(* IEC 61131-3 sources: std_i2980_v2.06_cp053/Source/IMM/ieccontrol/HostCommunication (part 2) *)

(* ---- FTimeToSec.pu ---- *)
(*
@h    ! WARNING !
@h    The Kemro K2 system (including software) only meets category B according to EN 954-1,
@h    thus it is not intended for usage in safety-relevant control applications in the field
@h    of personal safety (e.g. emergency stop).
@h    To implement potentially necessary safety-relevant control tasks, always use additional
@h    external safety devices that are intended for the particular purpose, and meet the necessary
@h    functional safety.
@h    For further information see EN 954-1 (EN ISO 13849-1) and/or the K2-x00 user manual, chapter
@h    "CE conformity, directives and standards".

returns a REAL value (unit s, precision 3 digits after point) for a TIME value

*)

FUNCTION FTimeToSec : REAL #DUMMY_EDIT_BLOCK

VAR_INPUT
 time : TIME;
END_VAR
#BEGIN_EDIT_BLOCK
(**************************************** WARNING ********************************************
 *** The KEBA Kemro K2 System including software is not intended for safety control tasks! ***
 ***                       For further information see Comment tab!                        ***
 *********************************************************************************************)

FTimeToSec := LINT_TO_REAL((TIME_TO_LINT(time)/1000))/1000.0;

;#END_EDIT_BLOCK END_FUNCTION

#END_OF_IEC_PART

@Puma @IecEditor 6 60 @Pou 25
@@@BEG_Comment@@@
@h    ! WARNING !
@h    The Kemro K2 system (including software) only meets category B according to EN 954-1,
@h    thus it is not intended for usage in safety-relevant control applications in the field
@h    of personal safety (e.g. emergency stop).
@h    To implement potentially necessary safety-relevant control tasks, always use additional
@h    external safety devices that are intended for the particular purpose, and meet the necessary
@h    functional safety.
@h    For further information see EN 954-1 (EN ISO 13849-1) and/or the K2-x00 user manual, chapter
@h    "CE conformity, directives and standards".

returns a REAL value (unit s, precision 3 digits after point) for a TIME value

@@@END_Comment@@@

@BEG_Contents

@BEG_Func
@RT(17)FuncTreeContainer
0
@END_Func

@BEG_Const
@RT(18)ConstTreeContainer
0
@END_Const

@BEG_Export

@BEG_Kind
@FUNCTION @RT(10)FTimeToSec @STRUCTURED_TEXT
@RT(4)REAL @RT(0) @RT(0)
@END_Kind

@BEG_Dcl
@RT(16)DclTreeContainer
1
@Var @RT(4)time @RT(0) @T @F @DT @RT(4)TIME @RT(0) @T @T @BASIC 0 @F
@F @F
@T
@BEG_Attrib
3 @RT(0) @RT(0) @RT(0)
@END_Attrib
1 1 @F @F @F @F

@END_Dcl

@END_Export

@BEG_Body
@TL(7)
(**************************************** WARNING ********************************************
 *** The KEBA Kemro K2 System including software is not intended for safety control tasks! ***
 ***                       For further information see Comment tab!                        ***
 *********************************************************************************************)

FTimeToSec := LINT_TO_REAL((TIME_TO_LINT(time)/1000))/1000.0;

@END_Body

@END_Contents

(* ---- ABEM63.pu ---- *)
(*
@h    ! WARNING !
@h    The Kemro K2 system (including software) only meets category B according to EN 954-1,
@h    thus it is not intended for usage in safety-relevant control applications in the field
@h    of personal safety (e.g. emergency stop).
@h    To implement potentially necessary safety-relevant control tasks, always use additional
@h    external safety devices that are intended for the particular purpose, and meet the necessary
@h    functional safety.
@h    For further information see EN 954-1 (EN ISO 13849-1) and/or the K2-x00 user manual, chapter
@h    "CE conformity, directives and standards".

Euromap63 specific application parameters
*)

IMPORT_OVER_LISTFILE
 STOP_PROCESS_ALGORITHM
, GET_SYNC_REFTO
, ASCII_TO_STRING
, cMaxInjectionUnits
, cMaxZones
, tsEM63
, tnOperationMode
, ABHeatingState

END_IMPORT

ALGORITHM_BLOCK ABEM63 #DUMMY_EDIT_BLOCK

SYSTEM_VAR
 sv_EM63 : tsEM63;
 sv_iPendingAlarms : DINT (* number of alarms pending with class 1,2,3 *);
 sv_OperationMode : tnOperationMode;
 sv_bBadPart : BOOL;
 sv_iShotCounterRetain : UDINT (* shot counter retain (used for lubrication) *);
 sv_bInitDone : BOOL (* IEC initialisation is finished (after movement registration) *);
END_VAR

SYSTEM_OBJECT
 TaskVis : TASK;
 PU_Task_7 : TASK;
END_OBJECT

VAR
 mbLastCycleBad : BOOL;
 mpiTrigger : REFTO UDINT;
END_VAR

POSTUPDATE_ALGORITHM pActivate ON TaskVis WITH sv_bInitDone,sv_EM63.bActivate

#BEGIN_EDIT_BLOCK
(**************************************** WARNING ********************************************
 *** The KEBA Kemro K2 System including software is not intended for safety control tasks! ***
 ***                       For further information see Comment tab!                        ***
 *********************************************************************************************)

IF (sv_EM63.bActivate AND sv_bInitDone) THEN
    mpiTrigger := @sv_iShotCounterRetain;
    START_PROCESS_ALGORITHM(paRun);
ELSE
    mpiTrigger := EMPTY;
    STOP_PROCESS_ALGORITHM(paRun);
END_IF;

;#END_EDIT_BLOCK END_ALGORITHM

ALGORITHM aMachineStatus

VAR
 bAlarms : BOOL;
 sMachineMode : STRING(2);
 bActStsChanged : BOOL;
 oldOpMode : tnOperationMode;
 oldAlarms : BOOL;
 oldCycleBad : BOOL;
 bInit : BOOL;
END_VAR
#BEGIN_EDIT_BLOCK
(**************************************** WARNING ********************************************
 *** The KEBA Kemro K2 System including software is not intended for safety control tasks! ***
 ***                       For further information see Comment tab!                        ***
 *********************************************************************************************)

// ActStsMachine
bAlarms := sv_iPendingAlarms > 0;

bActStsChanged := (oldOpMode <> sv_OperationMode) OR (oldAlarms <> bAlarms) OR (oldCycleBad <> mbLastCycleBad);

oldOpMode := sv_OperationMode;
oldAlarms := bAlarms;
oldCycleBad := mbLastCycleBad;

IF (bActStsChanged OR (NOT bInit)) THEN
    bInit := TRUE;

    CASE (sv_OperationMode) OF
        nFullAutomatic: sMachineMode := "A";
        nHalfAutomatic: sMachineMode := "S";
        nManual: sMachineMode := "M";
        nSetup: sMachineMode := "U";
    ELSE
        sMachineMode := "0";
    END_CASE;

    sv_EM63.ActStsMachine := CONCAT("0", sMachineMode, "0", DINT_TO_STRING(BOOL_TO_DINT(mbLastCycleBad)),  DINT_TO_STRING(BOOL_TO_DINT(bAlarms)));
END_IF;

;#END_EDIT_BLOCK END_ALGORITHM

PROCESS_ALGORITHM paRun ON TaskVis

VAR
 iRedCnt : INT;
 abHeatingState : ABHeatingState;
END_VAR
#BEGIN_EDIT_BLOCK
(**************************************** WARNING ********************************************
 *** The KEBA Kemro K2 System including software is not intended for safety control tasks! ***
 ***                       For further information see Comment tab!                        ***
 *********************************************************************************************)

IF (iRedCnt = 0) THEN
   iRedCnt := 5;

   aMachineStatus();
   abHeatingState.aHeating(bEM63 := TRUE);
END_IF;

iRedCnt := iRedCnt - 1;

;#END_EDIT_BLOCK END_ALGORITHM

POSTUPDATE_ALGORITHM pShotCounter ON PU_Task_7(1) WITH mpiTrigger^

#BEGIN_EDIT_BLOCK
(**************************************** WARNING ********************************************
 *** The KEBA Kemro K2 System including software is not intended for safety control tasks! ***
 ***                       For further information see Comment tab!                        ***
 *********************************************************************************************)

mbLastCycleBad := sv_bBadPart;

;#END_EDIT_BLOCK END_ALGORITHM

END_ALGORITHM_BLOCK

#END_OF_IEC_PART

@Puma @IecEditor 6 159 @Pou 25
@@@BEG_Comment@@@
@h    ! WARNING !
@h    The Kemro K2 system (including software) only meets category B according to EN 954-1,
@h    thus it is not intended for usage in safety-relevant control applications in the field
@h    of personal safety (e.g. emergency stop).
@h    To implement potentially necessary safety-relevant control tasks, always use additional
@h    external safety devices that are intended for the particular purpose, and meet the necessary
@h    functional safety.
@h    For further information see EN 954-1 (EN ISO 13849-1) and/or the K2-x00 user manual, chapter
@h    "CE conformity, directives and standards".

Euromap63 specific application parameters
@@@END_Comment@@@

@BEG_Contents

@BEG_Func
@RT(17)FuncTreeContainer
3
@Var @RT(22)STOP_PROCESS_ALGORITHM @RT(0) @T @T @DERIVED 0 @F @RT(23)KEBA_STANDARD_PROCEDURE @F
@T
@BEG_Attrib
0 @RT(0) @RT(0)
@END_Attrib
1 1 @F @F @F @F

@Var @RT(14)GET_SYNC_REFTO @RT(0) @T @T @DERIVED 0 @F @RT(22)KEBA_STANDARD_FUNCTION @F
@T
@BEG_Attrib
0 @RT(0) @RT(0)
@END_Attrib
1 1 @F @F @F @F

@Var @RT(15)ASCII_TO_STRING @RT(0) @T @T @DERIVED 0 @F @RT(22)KEBA_STANDARD_FUNCTION @F
@T
@BEG_Attrib
0 @RT(0) @RT(0)
@END_Attrib
1 1 @F @F @F @F

@END_Func

@BEG_Const
@RT(18)ConstTreeContainer
2
@Var @RT(18)cMaxInjectionUnits @RT(0) @T @F @DT @RT(4)DINT @RT(0) @T @T @BASIC 0 @F
@F @F
@T
@BEG_Attrib
0 @RT(1)2 @RT(0)
@END_Attrib
1 1 @F @F @F @F

@Var @RT(9)cMaxZones @RT(0) @T @F @DT @RT(4)DINT @RT(0) @T @T @BASIC 0 @F
@F @F
@T
@BEG_Attrib
0 @RT(2)72 @RT(27)max number of heating zones
@END_Attrib
1 1 @F @F @F @F

@END_Const

@BEG_Export

@BEG_Kind
@ALGORITHM_BLOCK @RT(6)ABEM63 @STRUCTURED_TEXT
@RT(0) @RT(0) @RT(0)
@END_Kind

@BEG_Dcl
@RT(16)DclTreeContainer
10
@Var @RT(7)sv_EM63 @RT(0) @T @T @DERIVED 0 @F @RT(6)tsEM63 @F
@T
@BEG_Attrib
3 @RT(0) @RT(0) @RT(0)
@END_Attrib
1 8 @F @F @F @F

@Var @RT(17)sv_iPendingAlarms @RT(0) @T @F @DT @RT(4)DINT @RT(0) @T @T @BASIC 0 @F
@F @F
@T
@BEG_Attrib
3 @RT(0) @RT(41)number of alarms pending with class 1,2,3 @RT(0)
@END_Attrib
1 8 @F @F @F @F

@Var @RT(16)sv_OperationMode @RT(0) @T @T @DERIVED 0 @T @T @DT @RT(15)tnOperationMode @RT(0) @T @T @UNKNOWN 0 @F
@F @F
@T
@BEG_Attrib
3 @RT(0) @RT(0) @RT(0)
@END_Attrib
1 8 @F @F @F @F

@Var @RT(11)sv_bBadPart @RT(0) @T @F @DT @RT(4)BOOL @RT(0) @T @T @BASIC 0 @F
@F @F
@T
@BEG_Attrib
3 @RT(0) @RT(0) @RT(0)
@END_Attrib
1 8 @F @F @F @F

@Var @RT(21)sv_iShotCounterRetain @RT(0) @T @F @DT @RT(5)UDINT @RT(0) @T @T @BASIC 0 @F
@F @F
@T
@BEG_Attrib
3 @RT(0) @RT(42)shot counter retain (used for lubrication) @RT(0)
@END_Attrib
1 8 @F @F @F @F

@Var @RT(12)sv_bInitDone @RT(0) @T @F @DT @RT(4)BOOL @RT(0) @T @T @BASIC 0 @F
@F @F
@T
@BEG_Attrib
3 @RT(0) @RT(60)IEC initialisation is finished (after movement registration) @RT(0)
@END_Attrib
1 8 @F @F @F @F

@Var @RT(7)TaskVis @RT(0) @T @T @RENAMED 0 @T @T @DT @RT(4)TASK @RT(0) @T @T @BASIC 0 @F
@F @F
@T
@BEG_Attrib
3 @RT(0) @RT(0) @RT(0)
@END_Attrib
1 7 @F @F @F @F

@Var @RT(9)PU_Task_7 @RT(0) @T @T @RENAMED 0 @T @T @DT @RT(4)TASK @RT(0) @T @T @BASIC 0 @F
@F @F
@T
@BEG_Attrib
3 @RT(0) @RT(0) @RT(0)
@END_Attrib
1 7 @F @F @F @F

@Var @RT(14)mbLastCycleBad @RT(0) @T @F @DT @RT(4)BOOL @RT(0) @T @T @BASIC 0 @F
@F @F
@T
@BEG_Attrib
3 @RT(0) @RT(0) @RT(0)
@END_Attrib
1 0 @F @F @F @F

@Var @RT(10)mpiTrigger @RT(0) @T @T @REFTO 0 @T @DT @RT(5)UDINT @RT(0) @T @T @BASIC 0 @F
@F @F
@T
@BEG_Attrib
3 @RT(0) @RT(0) @RT(0)
@END_Attrib
1 0 @F @F @F @F

@END_Dcl

@END_Export

@BEG_Body

4

@BEG_Export

@BEG_Algo
@POSTUPDATE_ALGORITHM @RT(9)pActivate @STRUCTURED_TEXT
@RT(0) @RT(30)sv_bInitDone,sv_EM63.bActivate @RT(7)TaskVis @F @F
@END_Algo

@BEG_Dcl
@RT(16)DclTreeContainer
0
@END_Dcl

@END_Export

@BEG_Export

@BEG_Algo
@ALGORITHM @RT(14)aMachineStatus @STRUCTURED_TEXT
@RT(0) @RT(0) @RT(0) @F @F
@END_Algo

@BEG_Dcl
@RT(16)DclTreeContainer
7
@Var @RT(7)bAlarms @RT(0) @T @F @DT @RT(4)BOOL @RT(0) @T @T @BASIC 0 @F
@F @F
@T
@BEG_Attrib
3 @RT(0) @RT(0) @RT(0)
@END_Attrib
1 0 @F @F @F @F

@Var @RT(12)sMachineMode @RT(0) @T @F @DT @RT(9)STRING(2) @RT(0) @T @T @STRING 0 @F @RT(1)2 @F
@F @F
@T
@BEG_Attrib
3 @RT(0) @RT(0) @RT(0)
@END_Attrib
1 0 @F @F @F @F

@Var @RT(14)bActStsChanged @RT(0) @T @F @DT @RT(4)BOOL @RT(0) @T @T @BASIC 0 @F
@F @F
@T
@BEG_Attrib
3 @RT(0) @RT(0) @RT(0)
@END_Attrib
1 0 @F @F @F @F

@Var @RT(9)oldOpMode @RT(0) @T @T @DERIVED 0 @T @T @DT @RT(15)tnOperationMode @RT(0) @T @T @UNKNOWN 0 @F
@F @F
@T
@BEG_Attrib
3 @RT(0) @RT(0) @RT(0)
@END_Attrib
1 0 @F @F @F @F

@Var @RT(9)oldAlarms @RT(0) @T @F @DT @RT(4)BOOL @RT(0) @T @T @BASIC 0 @F
@F @F
@T
@BEG_Attrib
3 @RT(0) @RT(0) @RT(0)
@END_Attrib
1 0 @F @F @F @F

@Var @RT(11)oldCycleBad @RT(0) @T @F @DT @RT(4)BOOL @RT(0) @T @T @BASIC 0 @F
@F @F
@T
@BEG_Attrib
3 @RT(0) @RT(0) @RT(0)
@END_Attrib
1 0 @F @F @F @F

@Var @RT(5)bInit @RT(0) @T @F @DT @RT(4)BOOL @RT(0) @T @T @BASIC 0 @F
@F @F
@T
@BEG_Attrib
3 @RT(0) @RT(0) @RT(0)
@END_Attrib
1 0 @F @F @F @F

@END_Dcl

@END_Export

@BEG_Export

@BEG_Algo
@PROCESS_ALGORITHM @RT(5)paRun @STRUCTURED_TEXT
@RT(0) @RT(0) @RT(7)TaskVis @F @F
@END_Algo

@BEG_Dcl
@RT(16)DclTreeContainer
2
@Var @RT(7)iRedCnt @RT(0) @T @F @DT @RT(3)INT @RT(0) @T @T @BASIC 0 @F
@F @F
@T
@BEG_Attrib
3 @RT(0) @RT(0) @RT(0)
@END_Attrib
1 0 @F @F @F @F

@Var @RT(14)abHeatingState @RT(0) @T @T @DERIVED 0 @F @RT(14)ABHeatingState @F
@T
@BEG_Attrib
3 @RT(0) @RT(0) @RT(0)
@END_Attrib
1 0 @F @F @F @F

@END_Dcl

@END_Export

@BEG_Export

@BEG_Algo
@POSTUPDATE_ALGORITHM @RT(12)pShotCounter @STRUCTURED_TEXT
@RT(0) @RT(11)mpiTrigger^ @RT(12)PU_Task_7(1) @F @F
@END_Algo

@BEG_Dcl
@RT(16)DclTreeContainer
0
@END_Dcl

@END_Export

@BEG_Body
@TL(13)
(**************************************** WARNING ********************************************
 *** The KEBA Kemro K2 System including software is not intended for safety control tasks! ***
 ***                       For further information see Comment tab!                        ***
 *********************************************************************************************)

IF (sv_EM63.bActivate AND sv_bInitDone) THEN
    mpiTrigger := @sv_iShotCounterRetain;
    START_PROCESS_ALGORITHM(paRun);
ELSE
    mpiTrigger := EMPTY;
    STOP_PROCESS_ALGORITHM(paRun);
END_IF;

@END_Body

@@@BEG_Comment@@@
@TL(0)

@@@END_Comment@@@

@BEG_Body
@TL(30)
(**************************************** WARNING ********************************************
 *** The KEBA Kemro K2 System including software is not intended for safety control tasks! ***
 ***                       For further information see Comment tab!                        ***
 *********************************************************************************************)

// ActStsMachine
bAlarms := sv_iPendingAlarms > 0;

bActStsChanged := (oldOpMode <> sv_OperationMode) OR (oldAlarms <> bAlarms) OR (oldCycleBad <> mbLastCycleBad);

oldOpMode := sv_OperationMode;
oldAlarms := bAlarms;
oldCycleBad := mbLastCycleBad;

IF (bActStsChanged OR (NOT bInit)) THEN
    bInit := TRUE;

    CASE (sv_OperationMode) OF
        nFullAutomatic: sMachineMode := "A";
        nHalfAutomatic: sMachineMode := "S";
        nManual: sMachineMode := "M";
        nSetup: sMachineMode := "U";
    ELSE
        sMachineMode := "0";
    END_CASE;

    sv_EM63.ActStsMachine := CONCAT("0", sMachineMode, "0", DINT_TO_STRING(BOOL_TO_DINT(mbLastCycleBad)),  DINT_TO_STRING(BOOL_TO_DINT(bAlarms)));
END_IF;

@END_Body

@@@BEG_Comment@@@
@TL(0)

@@@END_Comment@@@

@BEG_Body
@TL(14)
(**************************************** WARNING ********************************************
 *** The KEBA Kemro K2 System including software is not intended for safety control tasks! ***
 ***                       For further information see Comment tab!                        ***
 *********************************************************************************************)

IF (iRedCnt = 0) THEN
   iRedCnt := 5;

   aMachineStatus();
   abHeatingState.aHeating(bEM63 := TRUE);
END_IF;

iRedCnt := iRedCnt - 1;

@END_Body

@@@BEG_Comment@@@
@TL(0)

@@@END_Comment@@@

@BEG_Body
@TL(7)
(**************************************** WARNING ********************************************
 *** The KEBA Kemro K2 System including software is not intended for safety control tasks! ***
 ***                       For further information see Comment tab!                        ***
 *********************************************************************************************)

mbLastCycleBad := sv_bBadPart;

@END_Body

@@@BEG_Comment@@@
@TL(0)

@@@END_Comment@@@
@END_Body

@END_Contents

(* ---- ABEM77.pu ---- *)
IMPORT_OVER_LISTFILE
 KCAT_GetHandle
, ASSERT
, KMSG_SetProtocolVariable
, KCAT_GetValue
, tsEM77
, KCAT_HandleData
, KCAT_Status
, KMSG_Status
, ABHeatingState

END_IMPORT

ALGORITHM_BLOCK ABEM77 #DUMMY_EDIT_BLOCK

SYSTEM_VAR
 sv_EM77 : tsEM77;
 sv_bInitDone : BOOL (* IEC initialisation is finished (after movement registration) *);
 sv_bInitStart : BOOL;
END_VAR

SYSTEM_OBJECT
 PU_Task_7 : TASK;
 erAssert : ALARM;
 TaskVis : TASK;
END_OBJECT

POSTUPDATE_ALGORITHM pAvailable ON PU_Task_7 WITH sv_bInitStart,sv_EM77.bAvailable

VAR_TEMP
 hdlData : KCAT_HandleData;
 dummy : DINT;
 sProtocolVar : STRING(255);
 s : KCAT_Status;
 s2 : KMSG_Status;
 b : BOOL;
 i : INT;
 iMsgClass : DINT;
END_VAR

VAR
 msgClassFound : DWORD := 16#18020000;
END_VAR
#BEGIN_EDIT_BLOCK
(**************************************** WARNING ********************************************
 *** The KEBA Kemro K2 System including software is not intended for safety control tasks! ***
 ***                       For further information see Comment tab!                        ***
 *********************************************************************************************)

IF (sv_EM77.bAvailable AND sv_bInitStart) THEN
    // register protocol variable
    hdlData := KCAT_GetHandle("ILOG.varName");
    IF (hdlData.Status <> KCAT_Status_OK) THEN
        dummy := Print("ABEM77 Configuration problem: Production Counter for infolog not configured: ILOG.varName");
        b := ASSERT(FALSE, erAssert);
    END_IF;

    s := KCAT_GetValue(hdlData.Handle, sProtocolVar);
    IF (s <> KCAT_Status_OK) THEN
        dummy := Print("ABEM77 Configuration problem: cannot read ILOG.varName");
        b := ASSERT(FALSE, erAssert);
    END_IF;

    s2 := KMSG_SetProtocolVariable(CONCAT("APPL.", sProtocolVar));
    IF (s2 <> KMSG_Status_OK) THEN
        dummy := Print("ABEM77: cannot set variable ILOG.varName=%s as protocolvariable", sProtocolVar);
        b := ASSERT(FALSE, erAssert);
    END_IF;

    // check repsys config
    FOR i := 1 TO 32 DO
        hdlData := KCAT_GetHandle(CONCAT("RepSys.MsgClass:", INT_TO_STRING(i-1), ".msgClassNr"));
        IF (hdlData.Status = KCAT_Status_OK) THEN
              s := KCAT_GetValue(hdlData.Handle, iMsgClass);
              IF (s = KCAT_Status_OK) THEN
                  msgClassFound := msgClassFound AND (NOT (SHL(1, iMsgClass)));
                  IF (msgClassFound = 0) THEN
                      EXIT;
                  END_IF;
              END_IF;
        END_IF;
    END_FOR;

    IF (msgClassFound <> 0) THEN
        dummy := Print("ABEM77: Configuration problem - not all necessary RepSys classes configured!");
        b := ASSERT(FALSE, erAssert);
    END_IF;

END_IF;

;#END_EDIT_BLOCK END_ALGORITHM

POSTUPDATE_ALGORITHM pActivate ON TaskVis WITH sv_bInitDone,sv_EM77.bActivate

#BEGIN_EDIT_BLOCK
(**************************************** WARNING ********************************************
 *** The KEBA Kemro K2 System including software is not intended for safety control tasks! ***
 ***                       For further information see Comment tab!                        ***
 *********************************************************************************************)

IF (sv_EM77.bActivate AND sv_bInitDone) THEN
    START_PROCESS_ALGORITHM(paRun);
ELSE
    STOP_PROCESS_ALGORITHM(paRun);
END_IF;

;#END_EDIT_BLOCK END_ALGORITHM

PROCESS_ALGORITHM paRun ON TaskVis

VAR
 iRedCnt : INT;
 abHeatingState : ABHeatingState;
END_VAR
#BEGIN_EDIT_BLOCK
(**************************************** WARNING ********************************************
 *** The KEBA Kemro K2 System including software is not intended for safety control tasks! ***
 ***                       For further information see Comment tab!                        ***
 *********************************************************************************************)

IF (iRedCnt = 0) THEN
   iRedCnt := 5;

   abHeatingState.aHeating(bEM63 := TRUE);
END_IF;

iRedCnt := iRedCnt - 1;

;#END_EDIT_BLOCK END_ALGORITHM

END_ALGORITHM_BLOCK

#END_OF_IEC_PART

@Puma @IecEditor 6 179 @Pou 25
@@@BEG_Comment@@@

@@@END_Comment@@@

@BEG_Contents

@BEG_Func
@RT(17)FuncTreeContainer
4
@Var @RT(14)KCAT_GetHandle @RT(0) @T @F @DT @RT(0) @RT(0) @T @T @UNKNOWN 0 @F
@F @F
@T
@BEG_Attrib
0 @RT(0) @RT(0)
@END_Attrib
1 1 @F @F @F @F

@Var @RT(6)ASSERT @RT(0) @T @T @DERIVED 0 @F @RT(8)FUNCTION @F
@T
@BEG_Attrib
0 @RT(0) @RT(0)
@END_Attrib
1 1 @F @F @F @F

@Var @RT(24)KMSG_SetProtocolVariable @RT(0) @T @F @DT @RT(0) @RT(0) @T @T @UNKNOWN 0 @F
@F @F
@T
@BEG_Attrib
0 @RT(0) @RT(0)
@END_Attrib
1 1 @F @F @F @F

@Var @RT(13)KCAT_GetValue @RT(0) @T @F @DT @RT(0) @RT(0) @T @T @UNKNOWN 0 @F
@F @F
@T
@BEG_Attrib
0 @RT(0) @RT(0)
@END_Attrib
1 1 @F @F @F @F

@END_Func

@BEG_Const
@RT(18)ConstTreeContainer
0
@END_Const

@BEG_Export

@BEG_Kind
@ALGORITHM_BLOCK @RT(6)ABEM77 @STRUCTURED_TEXT
@RT(0) @RT(0) @RT(0)
@END_Kind

@BEG_Dcl
@RT(16)DclTreeContainer
6
@Var @RT(7)sv_EM77 @RT(0) @T @T @DERIVED 0 @T @T @DT @RT(6)tsEM77 @RT(0) @T @T @UNKNOWN 0 @F
@F @F
@T
@BEG_Attrib
3 @RT(0) @RT(0) @RT(0)
@END_Attrib
1 8 @F @F @F @F

@Var @RT(12)sv_bInitDone @RT(0) @T @F @DT @RT(4)BOOL @RT(0) @T @T @BASIC 0 @F
@F @F
@T
@BEG_Attrib
3 @RT(0) @RT(60)IEC initialisation is finished (after movement registration) @RT(0)
@END_Attrib
1 8 @F @F @F @F

@Var @RT(13)sv_bInitStart @RT(0) @T @T @RENAMED 0 @T @T @DT @RT(4)BOOL @RT(0) @T @T @BASIC 0 @F
@F @F
@T
@BEG_Attrib
3 @RT(0) @RT(0) @RT(0)
@END_Attrib
1 8 @F @F @F @F

@Var @RT(9)PU_Task_7 @RT(0) @T @T @RENAMED 0 @T @T @DT @RT(4)TASK @RT(0) @T @T @BASIC 0 @F
@F @F
@T
@BEG_Attrib
3 @RT(0) @RT(0) @RT(0)
@END_Attrib
1 7 @F @F @F @F

@Var @RT(8)erAssert @RT(0) @T @F @DT @RT(5)ALARM @RT(0) @T @T @BASIC 0 @F
@F @F
@T
@BEG_Attrib
3 @RT(0) @RT(0) @RT(0)
@END_Attrib
1 7 @F @F @F @F

@Var @RT(7)TaskVis @RT(0) @T @T @RENAMED 0 @T @T @DT @RT(4)TASK @RT(0) @T @T @BASIC 0 @F
@F @F
@T
@BEG_Attrib
3 @RT(0) @RT(0) @RT(0)
@END_Attrib
1 7 @F @F @F @F

@END_Dcl

@END_Export

@BEG_Body

3

@BEG_Export

@BEG_Algo
@POSTUPDATE_ALGORITHM @RT(10)pAvailable @STRUCTURED_TEXT
@RT(0) @RT(32)sv_bInitStart,sv_EM77.bAvailable @RT(9)PU_Task_7 @F @F
@END_Algo

@BEG_Dcl
@RT(16)DclTreeContainer
9
@Var @RT(7)hdlData @RT(0) @T @T @DERIVED 0 @T @T @DT @RT(15)KCAT_HandleData @RT(0) @T @T @UNKNOWN 0 @F
@F @F
@T
@BEG_Attrib
3 @RT(0) @RT(0) @RT(0)
@END_Attrib
1 4 @F @F @F @F

@Var @RT(5)dummy @RT(0) @T @F @DT @RT(4)DINT @RT(0) @T @T @BASIC 0 @F
@F @F
@T
@BEG_Attrib
3 @RT(0) @RT(0) @RT(0)
@END_Attrib
1 4 @F @F @F @F

@Var @RT(12)sProtocolVar @RT(0) @T @F @DT @RT(11)STRING(255) @RT(0) @T @T @STRING 0 @F @RT(3)255 @F
@F @F
@T
@BEG_Attrib
3 @RT(0) @RT(0) @RT(0)
@END_Attrib
1 4 @F @F @F @F

@Var @RT(1)s @RT(0) @T @T @DERIVED 0 @T @T @DT @RT(11)KCAT_Status @RT(0) @T @T @UNKNOWN 0 @F
@F @F
@T
@BEG_Attrib
3 @RT(0) @RT(0) @RT(0)
@END_Attrib
1 4 @F @F @F @F

@Var @RT(2)s2 @RT(0) @T @T @DERIVED 0 @T @T @DT @RT(11)KMSG_Status @RT(0) @T @T @UNKNOWN 0 @F
@F @F
@T
@BEG_Attrib
3 @RT(0) @RT(0) @RT(0)
@END_Attrib
1 4 @F @F @F @F

@Var @RT(1)b @RT(0) @T @F @DT @RT(4)BOOL @RT(0) @T @T @BASIC 0 @F
@F @F
@T
@BEG_Attrib
3 @RT(0) @RT(0) @RT(0)
@END_Attrib
1 4 @F @F @F @F

@Var @RT(1)i @RT(0) @T @F @DT @RT(3)INT @RT(0) @T @T @BASIC 0 @F
@F @F
@T
@BEG_Attrib
3 @RT(0) @RT(0) @RT(0)
@END_Attrib
1 4 @F @F @F @F

@Var @RT(9)iMsgClass @RT(0) @T @F @DT @RT(4)DINT @RT(0) @T @T @BASIC 0 @F
@F @F
@T
@BEG_Attrib
3 @RT(0) @RT(0) @RT(0)
@END_Attrib
1 4 @F @F @F @F

@Var @RT(13)msgClassFound @RT(0) @T @F @DT @RT(5)DWORD @RT(0) @T @T @BASIC 0 @F
@F @F
@T
@BEG_Attrib
3 @RT(11)16#18020000 @RT(0) @RT(0)
@END_Attrib
1 0 @F @F @F @F

@END_Dcl

@END_Export

@BEG_Export

@BEG_Algo
@POSTUPDATE_ALGORITHM @RT(9)pActivate @STRUCTURED_TEXT
@RT(0) @RT(30)sv_bInitDone,sv_EM77.bActivate @RT(7)TaskVis @F @F
@END_Algo

@BEG_Dcl
@RT(16)DclTreeContainer
0
@END_Dcl

@END_Export

@BEG_Export

@BEG_Algo
@PROCESS_ALGORITHM @RT(5)paRun @STRUCTURED_TEXT
@RT(0) @RT(0) @RT(7)TaskVis @F @F
@END_Algo

@BEG_Dcl
@RT(16)DclTreeContainer
2
@Var @RT(7)iRedCnt @RT(0) @T @F @DT @RT(3)INT @RT(0) @T @T @BASIC 0 @F
@F @F
@T
@BEG_Attrib
3 @RT(0) @RT(0) @RT(0)
@END_Attrib
1 0 @F @F @F @F

@Var @RT(14)abHeatingState @RT(0) @T @T @DERIVED 0 @T @T @DT @RT(14)ABHeatingState @RT(0) @T @T @UNKNOWN 0 @F
@F @F
@T
@BEG_Attrib
3 @RT(0) @RT(0) @RT(0)
@END_Attrib
1 0 @F @F @F @F

@END_Dcl

@END_Export

@BEG_Body
@TL(46)
(**************************************** WARNING ********************************************
 *** The KEBA Kemro K2 System including software is not intended for safety control tasks! ***
 ***                       For further information see Comment tab!                        ***
 *********************************************************************************************)

IF (sv_EM77.bAvailable AND sv_bInitStart) THEN
    // register protocol variable
    hdlData := KCAT_GetHandle("ILOG.varName");
    IF (hdlData.Status <> KCAT_Status_OK) THEN
        dummy := Print("ABEM77 Configuration problem: Production Counter for infolog not configured: ILOG.varName");
        b := ASSERT(FALSE, erAssert);
    END_IF;

    s := KCAT_GetValue(hdlData.Handle, sProtocolVar);
    IF (s <> KCAT_Status_OK) THEN
        dummy := Print("ABEM77 Configuration problem: cannot read ILOG.varName");
        b := ASSERT(FALSE, erAssert);
    END_IF;

    s2 := KMSG_SetProtocolVariable(CONCAT("APPL.", sProtocolVar));
    IF (s2 <> KMSG_Status_OK) THEN
        dummy := Print("ABEM77: cannot set variable ILOG.varName=%s as protocolvariable", sProtocolVar);
        b := ASSERT(FALSE, erAssert);
    END_IF;

    // check repsys config
    FOR i := 1 TO 32 DO
        hdlData := KCAT_GetHandle(CONCAT("RepSys.MsgClass:", INT_TO_STRING(i-1), ".msgClassNr"));
        IF (hdlData.Status = KCAT_Status_OK) THEN
              s := KCAT_GetValue(hdlData.Handle, iMsgClass);
              IF (s = KCAT_Status_OK) THEN
                  msgClassFound := msgClassFound AND (NOT (SHL(1, iMsgClass)));
                  IF (msgClassFound = 0) THEN
                      EXIT;
                  END_IF;
              END_IF;
        END_IF;
    END_FOR;

    IF (msgClassFound <> 0) THEN
        dummy := Print("ABEM77: Configuration problem - not all necessary RepSys classes configured!");
        b := ASSERT(FALSE, erAssert);
    END_IF;

END_IF;

@END_Body

@@@BEG_Comment@@@
@TL(0)

@@@END_Comment@@@

@BEG_Body
@TL(11)
(**************************************** WARNING ********************************************
 *** The KEBA Kemro K2 System including software is not intended for safety control tasks! ***
 ***                       For further information see Comment tab!                        ***
 *********************************************************************************************)

IF (sv_EM77.bActivate AND sv_bInitDone) THEN
    START_PROCESS_ALGORITHM(paRun);
ELSE
    STOP_PROCESS_ALGORITHM(paRun);
END_IF;

@END_Body

@@@BEG_Comment@@@
@TL(0)

@@@END_Comment@@@

@BEG_Body
@TL(13)
(**************************************** WARNING ********************************************
 *** The KEBA Kemro K2 System including software is not intended for safety control tasks! ***
 ***                       For further information see Comment tab!                        ***
 *********************************************************************************************)

IF (iRedCnt = 0) THEN
   iRedCnt := 5;

   abHeatingState.aHeating(bEM63 := TRUE);
END_IF;

iRedCnt := iRedCnt - 1;

@END_Body

@@@BEG_Comment@@@
@TL(0)

@@@END_Comment@@@
@END_Body

@END_Contents

(* ---- ABHostCom.pu ---- *)
(*
@h    ! WARNING !
@h    The Kemro K2 system (including software) only meets category B according to EN 954-1,
@h    thus it is not intended for usage in safety-relevant control applications in the field
@h    of personal safety (e.g. emergency stop).
@h    To implement potentially necessary safety-relevant control tasks, always use additional
@h    external safety devices that are intended for the particular purpose, and meet the necessary
@h    functional safety.
@h    For further information see EN 954-1 (EN ISO 13849-1) and/or the K2-x00 user manual, chapter
@h    "CE conformity, directives and standards".
*)

IMPORT_OVER_LISTFILE
 FHostTypeToString
, GET_TASK_INTERVAL
, FCreateHostComVersion
, cHostTypeNone
, cHostTypeOPCUA_EM77
, tsHostHmi
, tsHostCom
, tsEM77
, tsEM63
, KPROT_Status

END_IMPORT

ALGORITHM_BLOCK ABHostCom #DUMMY_EDIT_BLOCK

SYSTEM_VAR
 sv_HostHmi : tsHostHmi;
 sv_bHostAvailable : BOOL;
 sv_HostCom : tsHostCom;
 sv_bInitDone : BOOL (* IEC initialisation is finished (after movement registration) *);
 sv_EM77 : tsEM77;
 sv_EM63 : tsEM63;
END_VAR

SYSTEM_OBJECT
 TaskVis : TASK;
END_OBJECT

VAR
 msILog : STRING(128);
END_VAR

(*
@h    ! WARNING !
@h    The Kemro K2 system (including software) only meets category B according to EN 954-1,
@h    thus it is not intended for usage in safety-relevant control applications in the field
@h    of personal safety (e.g. emergency stop).
@h    To implement potentially necessary safety-relevant control tasks, always use additional
@h    external safety devices that are intended for the particular purpose, and meet the necessary
@h    functional safety.
@h    For further information see EN 954-1 (EN ISO 13849-1) and/or the K2-x00 user manual, chapter
@h    "CE conformity, directives and standards".

connection supervision

*)

PROCESS_ALGORITHM paCheckConnection ON TaskVis AUTOSTART

VAR
 iStep : DINT;
 cycleTime : TIME;
 timeOutCnt : DINT;
 b : BOOL;
END_VAR

VAR CONSTANT
 connectionTimeout : TIME := T#30s;
END_VAR
#BEGIN_EDIT_BLOCK
(**************************************** WARNING ********************************************
 *** The KEBA Kemro K2 System including software is not intended for safety control tasks! ***
 ***                       For further information see Comment tab!                        ***
 *********************************************************************************************)

// Init Step
IF iStep = 0 THEN
   b := FCreateHostComVersion();
   cycleTime := GET_TASK_INTERVAL();
   iStep := 10;
END_IF;

// not connected step
IF iStep = 10 THEN
   sv_HostHmi.bIsConnected := FALSE;
   IF (sv_HostCom.bConnect AND (sv_HostCom.iHostTypeId <> cHostTypeNone) AND sv_bInitDone) THEN
      IF (sv_HostCom.iHostTypeId = cHostTypeOPC_EM63) THEN
         sv_EM63.bActivate := TRUE;
      ELSIF (sv_HostCom.iHostTypeId = cHostTypeOPCUA_EM77) THEN
         sv_EM77.bAvailable := TRUE;
         sv_EM77.bActivate := TRUE;
      END_IF;
      iStep := 20;
   END_IF;
END_IF;

// connected step
IF iStep = 20 THEN
   sv_HostHmi.bIsConnected := TRUE;

   sv_HostCom.bConnect := FALSE;
   timeOutCnt := LINT_TO_DINT(TIME_TO_LINT(connectionTimeout) / TIME_TO_LINT(cycleTime));
   iStep := 30;
END_IF;

// wait for connected bit
IF iStep = 30 THEN
   timeOutCnt := timeOutCnt - 1;
   IF sv_HostCom.bConnect THEN
      iStep := 20;
   END_IF;
   IF timeOutCnt = 0 THEN
      iStep := 10;
   END_IF;
END_IF;

;#END_EDIT_BLOCK END_ALGORITHM

POSTUPDATE_ALGORITHM pLogHostConnected ON TaskVis WITH sv_HostHmi.bIsConnected

VAR
 s : KPROT_Status;
 sType : STRING(16);
END_VAR
#BEGIN_EDIT_BLOCK
sType := FHostTypeToString(sv_HostCom.iHostTypeId);
msILog := CONCAT("Control station of type ", DINT_TO_STRING(sv_HostCom.iHostTypeId), " (", sType, ") ");

IF (sv_HostHmi.bIsConnected) THEN
    sv_bHostAvailable := TRUE;
    msILog := CONCAT(msILog, "connected");
ELSE
    msILog := CONCAT(msILog, "disconnected");
END_IF;

s := KPROT_UserInfoLog("%5s", 100, BOOL_TO_DINT(sv_HostHmi.bIsConnected), sv_HostCom.iHostTypeId, 0, msILog);

;#END_EDIT_BLOCK END_ALGORITHM

END_ALGORITHM_BLOCK

#END_OF_IEC_PART

@Puma @IecEditor 6 114 @Pou 25
@@@BEG_Comment@@@
@h    ! WARNING !
@h    The Kemro K2 system (including software) only meets category B according to EN 954-1,
@h    thus it is not intended for usage in safety-relevant control applications in the field
@h    of personal safety (e.g. emergency stop).
@h    To implement potentially necessary safety-relevant control tasks, always use additional
@h    external safety devices that are intended for the particular purpose, and meet the necessary
@h    functional safety.
@h    For further information see EN 954-1 (EN ISO 13849-1) and/or the K2-x00 user manual, chapter
@h    "CE conformity, directives and standards".
@@@END_Comment@@@

@BEG_Contents

@BEG_Func
@RT(17)FuncTreeContainer
3
@Var @RT(17)FHostTypeToString @RT(0) @T @T @DERIVED 0 @F @RT(8)FUNCTION @F
@T
@BEG_Attrib
0 @RT(0) @RT(0)
@END_Attrib
1 1 @F @F @F @F

@Var @RT(17)GET_TASK_INTERVAL @RT(0) @T @T @DERIVED 0 @F @RT(22)KEBA_STANDARD_FUNCTION @F
@T
@BEG_Attrib
0 @RT(0) @RT(0)
@END_Attrib
1 1 @F @F @F @F

@Var @RT(21)FCreateHostComVersion @RT(0) @T @T @DERIVED 0 @F @RT(8)FUNCTION @F
@T
@BEG_Attrib
0 @RT(0) @RT(0)
@END_Attrib
1 1 @F @F @F @F

@END_Func

@BEG_Const
@RT(18)ConstTreeContainer
2
@Var @RT(13)cHostTypeNone @RT(0) @T @F @DT @RT(4)DINT @RT(0) @T @T @BASIC 0 @F
@F @F
@T
@BEG_Attrib
0 @RT(1)0 @RT(0)
@END_Attrib
1 1 @F @F @F @F

@Var @RT(19)cHostTypeOPCUA_EM77 @RT(0) @T @F @DT @RT(4)DINT @RT(0) @T @T @BASIC 0 @F
@F @F
@T
@BEG_Attrib
0 @RT(1)7 @RT(0)
@END_Attrib
1 1 @F @F @F @F

@END_Const

@BEG_Export

@BEG_Kind
@ALGORITHM_BLOCK @RT(9)ABHostCom @STRUCTURED_TEXT
@RT(0) @RT(0) @RT(0)
@END_Kind

@BEG_Dcl
@RT(16)DclTreeContainer
8
@Var @RT(7)TaskVis @RT(0) @T @F @DT @RT(4)TASK @RT(0) @T @T @BASIC 0 @F
@F @F
@T
@BEG_Attrib
3 @RT(0) @RT(0) @RT(0)
@END_Attrib
1 7 @F @F @F @F

@Var @RT(10)sv_HostHmi @RT(0) @T @T @DERIVED 0 @T @T @DT @RT(9)tsHostHmi @RT(0) @T @T @UNKNOWN 0 @F
@F @F
@T
@BEG_Attrib
3 @RT(0) @RT(0) @RT(0)
@END_Attrib
1 8 @F @F @F @F

@Var @RT(17)sv_bHostAvailable @RT(0) @T @F @DT @RT(4)BOOL @RT(0) @T @T @BASIC 0 @F
@F @F
@T
@BEG_Attrib
3 @RT(0) @RT(0) @RT(0)
@END_Attrib
1 8 @F @F @F @F

@Var @RT(10)sv_HostCom @RT(0) @T @T @DERIVED 0 @T @T @DT @RT(9)tsHostCom @RT(0) @T @T @UNKNOWN 0 @F
@F @F
@T
@BEG_Attrib
3 @RT(0) @RT(0) @RT(0)
@END_Attrib
1 8 @F @F @F @F

@Var @RT(12)sv_bInitDone @RT(0) @T @F @DT @RT(4)BOOL @RT(0) @T @T @BASIC 0 @F
@F @F
@T
@BEG_Attrib
3 @RT(0) @RT(60)IEC initialisation is finished (after movement registration) @RT(0)
@END_Attrib
1 8 @F @F @F @F

@Var @RT(6)msILog @RT(0) @T @F @DT @RT(11)STRING(128) @RT(0) @T @T @STRING 0 @F @RT(3)128 @F
@F @F
@T
@BEG_Attrib
3 @RT(0) @RT(0) @RT(0)
@END_Attrib
1 0 @F @F @F @F

@Var @RT(7)sv_EM77 @RT(0) @T @T @DERIVED 0 @T @T @DT @RT(6)tsEM77 @RT(0) @T @T @UNKNOWN 0 @F
@F @F
@T
@BEG_Attrib
3 @RT(0) @RT(0) @RT(0)
@END_Attrib
1 8 @F @F @F @F

@Var @RT(7)sv_EM63 @RT(0) @T @T @DERIVED 0 @T @T @DT @RT(6)tsEM63 @RT(0) @T @T @UNKNOWN 0 @F
@F @F
@T
@BEG_Attrib
3 @RT(0) @RT(0) @RT(0)
@END_Attrib
1 8 @F @F @F @F

@END_Dcl

@END_Export

@BEG_Body

2

@BEG_Export

@BEG_Algo
@PROCESS_ALGORITHM @RT(17)paCheckConnection @STRUCTURED_TEXT
@RT(0) @RT(0) @RT(7)TaskVis @T @F
@END_Algo

@BEG_Dcl
@RT(16)DclTreeContainer
5
@Var @RT(5)iStep @RT(0) @T @F @DT @RT(4)DINT @RT(0) @T @T @BASIC 0 @F
@F @F
@T
@BEG_Attrib
3 @RT(0) @RT(0) @RT(0)
@END_Attrib
1 0 @F @F @F @F

@Var @RT(9)cycleTime @RT(0) @T @F @DT @RT(4)TIME @RT(0) @T @T @BASIC 0 @F
@F @F
@T
@BEG_Attrib
3 @RT(0) @RT(0) @RT(0)
@END_Attrib
1 0 @F @F @F @F

@Var @RT(17)connectionTimeout @RT(0) @T @F @DT @RT(4)TIME @RT(0) @T @T @BASIC 0 @F
@F @F
@T
@BEG_Attrib
3 @RT(5)T#30s @RT(0) @RT(0)
@END_Attrib
1 15 @F @F @F @F

@Var @RT(10)timeOutCnt @RT(0) @T @F @DT @RT(4)DINT @RT(0) @T @T @BASIC 0 @F
@F @F
@T
@BEG_Attrib
3 @RT(0) @RT(0) @RT(0)
@END_Attrib
1 0 @F @F @F @F

@Var @RT(1)b @RT(0) @T @F @DT @RT(4)BOOL @RT(0) @T @T @BASIC 0 @F
@F @F
@T
@BEG_Attrib
3 @RT(0) @RT(0) @RT(0)
@END_Attrib
1 0 @F @F @F @F

@END_Dcl

@END_Export

@BEG_Export

@BEG_Algo
@POSTUPDATE_ALGORITHM @RT(17)pLogHostConnected @STRUCTURED_TEXT
@RT(0) @RT(23)sv_HostHmi.bIsConnected @RT(7)TaskVis @F @F
@END_Algo

@BEG_Dcl
@RT(16)DclTreeContainer
2
@Var @RT(1)s @RT(0) @T @T @DERIVED 0 @T @T @DT @RT(12)KPROT_Status @RT(0) @T @T @UNKNOWN 0 @F
@F @F
@T
@BEG_Attrib
3 @RT(0) @RT(0) @RT(0)
@END_Attrib
1 0 @F @F @F @F

@Var @RT(5)sType @RT(0) @T @F @DT @RT(10)STRING(16) @RT(0) @T @T @STRING 0 @F @RT(2)16 @F
@F @F
@T
@BEG_Attrib
3 @RT(0) @RT(0) @RT(0)
@END_Attrib
1 0 @F @F @F @F

@END_Dcl

@END_Export

@BEG_Body
@TL(51)
(**************************************** WARNING ********************************************
 *** The KEBA Kemro K2 System including software is not intended for safety control tasks! ***
 ***                       For further information see Comment tab!                        ***
 *********************************************************************************************)

// Init Step
IF iStep = 0 THEN
   b := FCreateHostComVersion();
   cycleTime := GET_TASK_INTERVAL();
   iStep := 10;
END_IF;

// not connected step
IF iStep = 10 THEN
   sv_HostHmi.bIsConnected := FALSE;
   IF (sv_HostCom.bConnect AND (sv_HostCom.iHostTypeId <> cHostTypeNone) AND sv_bInitDone) THEN
      IF (sv_HostCom.iHostTypeId = cHostTypeOPC_EM63) THEN
         sv_EM63.bActivate := TRUE;
      ELSIF (sv_HostCom.iHostTypeId = cHostTypeOPCUA_EM77) THEN
         sv_EM77.bAvailable := TRUE;
         sv_EM77.bActivate := TRUE;
      END_IF;
      iStep := 20;
   END_IF;
END_IF;

// connected step
IF iStep = 20 THEN
   sv_HostHmi.bIsConnected := TRUE;

   sv_HostCom.bConnect := FALSE;
   timeOutCnt := LINT_TO_DINT(TIME_TO_LINT(connectionTimeout) / TIME_TO_LINT(cycleTime));
   iStep := 30;
END_IF;

// wait for connected bit
IF iStep = 30 THEN
   timeOutCnt := timeOutCnt - 1;
   IF sv_HostCom.bConnect THEN
      iStep := 20;
   END_IF;
   IF timeOutCnt = 0 THEN
      iStep := 10;
   END_IF;
END_IF;

@END_Body

@@@BEG_Comment@@@
@TL(13)
@h    ! WARNING !
@h    The Kemro K2 system (including software) only meets category B according to EN 954-1,
@h    thus it is not intended for usage in safety-relevant control applications in the field
@h    of personal safety (e.g. emergency stop).
@h    To implement potentially necessary safety-relevant control tasks, always use additional
@h    external safety devices that are intended for the particular purpose, and meet the necessary
@h    functional safety.
@h    For further information see EN 954-1 (EN ISO 13849-1) and/or the K2-x00 user manual, chapter
@h    "CE conformity, directives and standards".

connection supervision

@@@END_Comment@@@

@BEG_Body
@TL(15)
sType := FHostTypeToString(sv_HostCom.iHostTypeId);
msILog := CONCAT("Control station of type ", DINT_TO_STRING(sv_HostCom.iHostTypeId), " (", sType, ") ");

IF (sv_HostHmi.bIsConnected) THEN
    sv_bHostAvailable := TRUE;
    msILog := CONCAT(msILog, "connected");
ELSE
    msILog := CONCAT(msILog, "disconnected");
END_IF;

s := KPROT_UserInfoLog("%5s", 100, BOOL_TO_DINT(sv_HostHmi.bIsConnected), sv_HostCom.iHostTypeId, 0, msILog);

@END_Body

@@@BEG_Comment@@@
@TL(0)

@@@END_Comment@@@
@END_Body

@END_Contents
